FUNCTION_BLOCK INTERNAL ABSTRACT POU_1
VAR_INPUT
END_VAR
VAR_OUTPUT
END_VAR
VAR
END_VAR

END_FUNCTION_BLOCK

(* stored: Version 1.1.0.1, ProductVersion 3.1.4024.12
   POU POU_1: Id {1e338645-51e7-4f1d-b0d1-2a20383756e8}, SpecialFunc None *)
